FUNCTION_BLOCK FB_SetValvesClose
VAR_INPUT
    fbValveNames : ARRAY[1..GVL.valveCount]OF STRING;
    fbNumValvesToPosition : INT;
END_VAR

VAR_IN_OUT
    fbValves : ARRAY[1..GVL.valveCount] OF ST_Valves;
END_VAR
VAR
    i : INT;
    j : INT;
END_VAR

FOR i := 1 TO fbNumValvesToPosition DO
    FOR j := 1 TO gvl.valveCount DO
        IF fbValves[j].name = fbValveNames[i] THEN
            fbValves[j].state := 0;
            fbValves[j].hOpenClose := FALSE;
            EXIT;
        END_IF
    END_FOR
END_FOR;

END_FUNCTION_BLOCK

(* stored: Version 1.1.0.1
   POU FB_SetValvesClose: Id {8d4d32fa-bcb8-0da0-3ed8-d40901c8979c}, SpecialFunc None *)
